// Mitsubishi GX Works2 project: Ex2   PLC: Q03UDV

PROGRAM MAIN
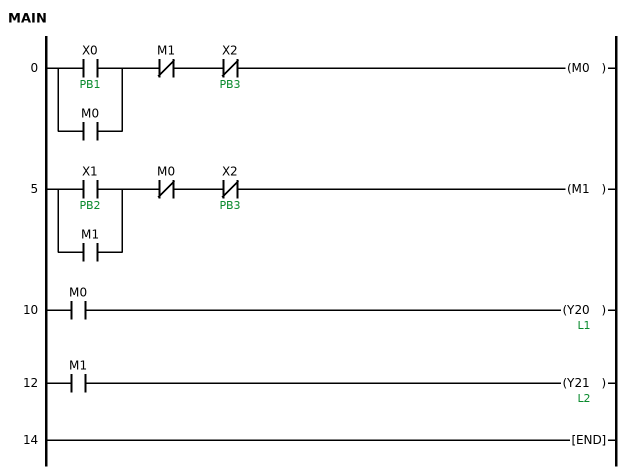
0     LD      X0  ; PB1
      OR      M0
      ANI     M1
      ANI     X2  ; PB3
      OUT     M0
5     LD      X1  ; PB2
      OR      M1
      ANI     M0
      ANI     X2  ; PB3
      OUT     M1
10    LD      M0
      OUT     Y20  ; L1
12    LD      M1
      OUT     Y21  ; L2
14    END
END_PROGRAM
